Universal Robots PolyScope program: swing.urp

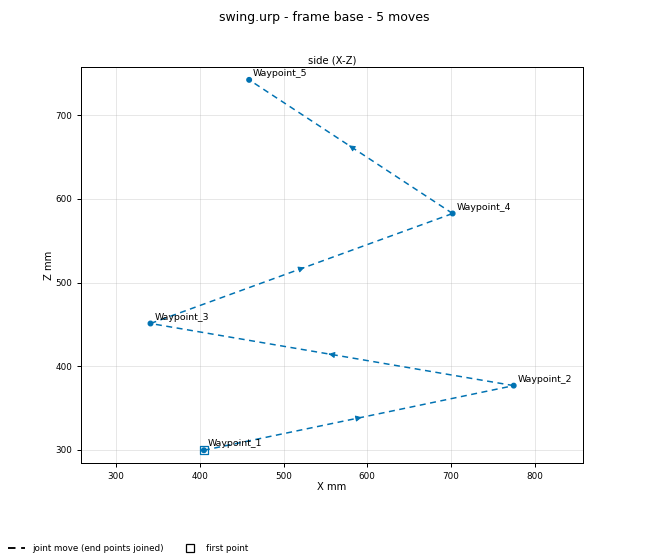
[picture p0: tool path of swing.urp in frame base, 5 of 5 moves have a stored position in this frame; points joined in program order, loops and branches not executed]
Program swing (installation=default directory=/programs createdIn=5.2.0.61336 lastSavedIn=5.2.0.61336 robotSerialNumber=20195500451)
Calibrated DH parameters: a=[0.00002, -0.231658, -0.317125, 0.000011, 0.000055, 0]; d=[0.162082, 123.190176, -180.284242, 57.22734, 0.099524, 0.09934]; alpha=[1.569304, 0.00289, 0.004025, 1.569925, -1.569026, 0]; deltaTheta=[0, 0.993923, 4.662183, 0.627072, 0.000001, 0]
Robot Program (runOnlyOnce=true)
  MoveJ speed 100 deg/s, acceleration 100 deg/s^2 (useActiveTCP=true) feature=Base
    Waypoint Waypoint_1: motionParameters(nextMotionTime=2); TCP in base x=404.825 y=-232.169 z=299.516 mm, rx=1.2321 ry=-1.1754 rz=1.1789 rad; joints [-0.002, -92.546, -130.073, -59.999, 0, 10.098] deg
    Waypoint Waypoint_2: motionParameters(nextMotionTime=0.5); TCP in base x=775.079 y=-233.354 z=376.757 mm, rx=1.224 ry=-1.1799 rz=1.1856 rad; joints [0, -135.326, -60.789, -59.999, 0.003, -15.915] deg
    Wait Sleep waitTime=0.3
    Waypoint Waypoint_3: motionParameters(nextMotionTime=0.5); TCP in base x=340.961 y=-231.996 z=451.011 mm, rx=1.2582 ry=-1.1296 rz=1.1351 rad; joints [0, -72.793, -127.261, -60.001, 0.003, -15.914] deg
    Wait Sleep waitTime=0.2
    Waypoint Waypoint_4: motionParameters(nextMotionTime=0.5); TCP in base x=702.088 y=-233.08 z=582.479 mm, rx=1.2119 ry=-1.1977 rz=1.2031 rad; joints [0, -122.047, -56.79, -60, 0.002, -31.81] deg
    Waypoint Waypoint_5: motionParameters(nextMotionTime=0.4 blendRadius=0.05); TCP in base x=458.884 y=-232.603 z=742.217 mm, rx=1.1103 ry=-1.3465 rz=1.3518 rad; joints [0.002, -90.539, -76.627, -59.999, 0.004, -31.81] deg
